FUNCTION F_UpdateParametersByReference
VAR_INPUT
	bSetNewValue : BOOL;
	fMaxPistonStroke : LREAL;
	paramCylinderPiston : REFERENCE TO ST_pPistonRange;
END_VAR
VAR
END_VAR

IF bSetNewValue THEN
	paramCylinderPiston.fPistonPosMax := fMaxPistonStroke;
	bSetNewValue := FALSE;
END_IF

END_FUNCTION

(* stored: Version 1.1.0.1, ProductVersion 3.1.4024.10
   POU F_UpdateParametersByReference: Id {a3b70210-cc9b-49fe-aa74-e453981806ae}, SpecialFunc None *)
